// Mitsubishi GX Works2 project: flash_LED   PLC: Q03UDV

PROGRAM MAIN
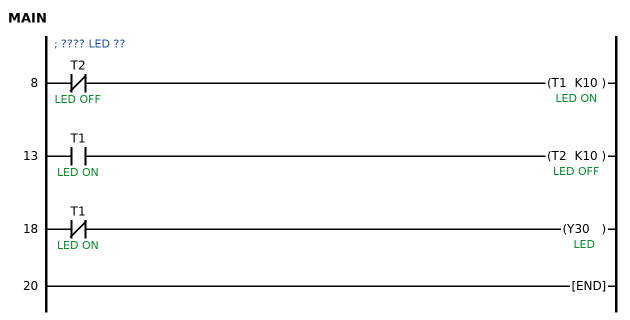
; ???? LED ??
8     LDI     T2  ; LED OFF
      OUT     T1 K10  ; LED ON
13    LD      T1  ; LED ON
      OUT     T2 K10  ; LED OFF
18    LDI     T1  ; LED ON
      OUT     Y30  ; LED
20    END
END_PROGRAM
